FUNCTION_BLOCK REAL2TIME_Feed (* Basic Function Block Type *)
  (* Standard: 61499-2 *)
  (* Version 0.0, 12/28/2023, SESA371406, Schneider Electric, Template *)
  PACKAGE SE.Nereda;
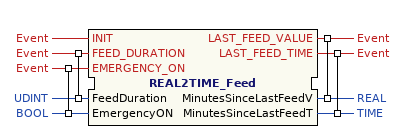
  EVENT_INPUT
    INIT;
    FEED_DURATION WITH FeedDuration;
    EMERGENCY_ON WITH EmergencyON;
  END_EVENT
  EVENT_OUTPUT
    LAST_FEED_VALUE WITH MinutesSinceLastFeedV; (* Execution Confirmation *)
    LAST_FEED_TIME WITH MinutesSinceLastFeedT;
  END_EVENT
  VAR_INPUT
    FeedDuration : UDINT; (* Input event qualifier *)
    EmergencyON : BOOL;
  END_VAR
  VAR_OUTPUT
    MinutesSinceLastFeedV : REAL := 1;
    MinutesSinceLastFeedT : TIME; (* Output event qualifier *)
  END_VAR
  VAR
    InValue : REAL;
  END_VAR
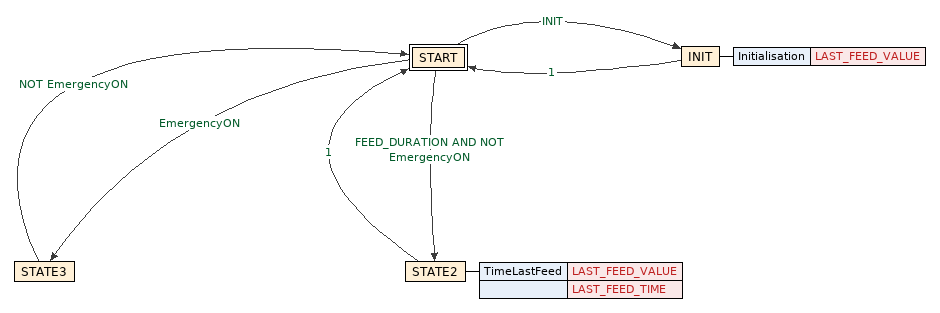
  EC_STATES
    START; (* Initial State *)
    STATE2 : TimeLastFeed -> LAST_FEED_VALUE, -> LAST_FEED_TIME; (* Initialization *)
    INIT : Initialisation -> LAST_FEED_VALUE;
    STATE3;
  END_STATES
  EC_TRANSITIONS
    START TO STATE2 := FEED_DURATION AND NOT EmergencyON;
    STATE2 TO START := 1;
    START TO INIT := INIT;
    INIT TO START := 1;
    START TO STATE3 := EmergencyON;
    STATE3 TO START := NOT EmergencyON;
  END_TRANSITIONS
  ALGORITHM TimeLastFeed IN ST: (* Initialization algorithm *)
;
// Convert real to time

InValue := UDINT_TO_REAL(FeedDuration) * 1000;
MinutesSinceLastFeedT := REAL_TO_TIME(InValue);
MinutesSinceLastFeedV := InValue / 1000;
  END_ALGORITHM
  ALGORITHM Initialisation IN ST:
;
MinutesSinceLastFeedV := 1.0;
  END_ALGORITHM
END_FUNCTION_BLOCK
